SUBAPPLICATION Automatik (* Subapplication Type *)
  (* Standard: 61499-2 *)
  (* Version 1.0, 2023-01-29, Franz *)
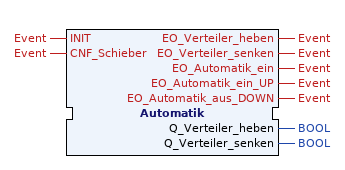
  EVENT_INPUT
    INIT;
    CNF_Schieber;
  END_EVENT
  EVENT_OUTPUT
    EO_Verteiler_heben;
    EO_Verteiler_senken;
    EO_Automatik_ein;
    EO_Automatik_ein_UP;
    EO_Automatik_aus_DOWN;
  END_EVENT
  VAR_OUTPUT
    Q_Verteiler_heben : BOOL;
    Q_Verteiler_senken : BOOL;
  END_VAR
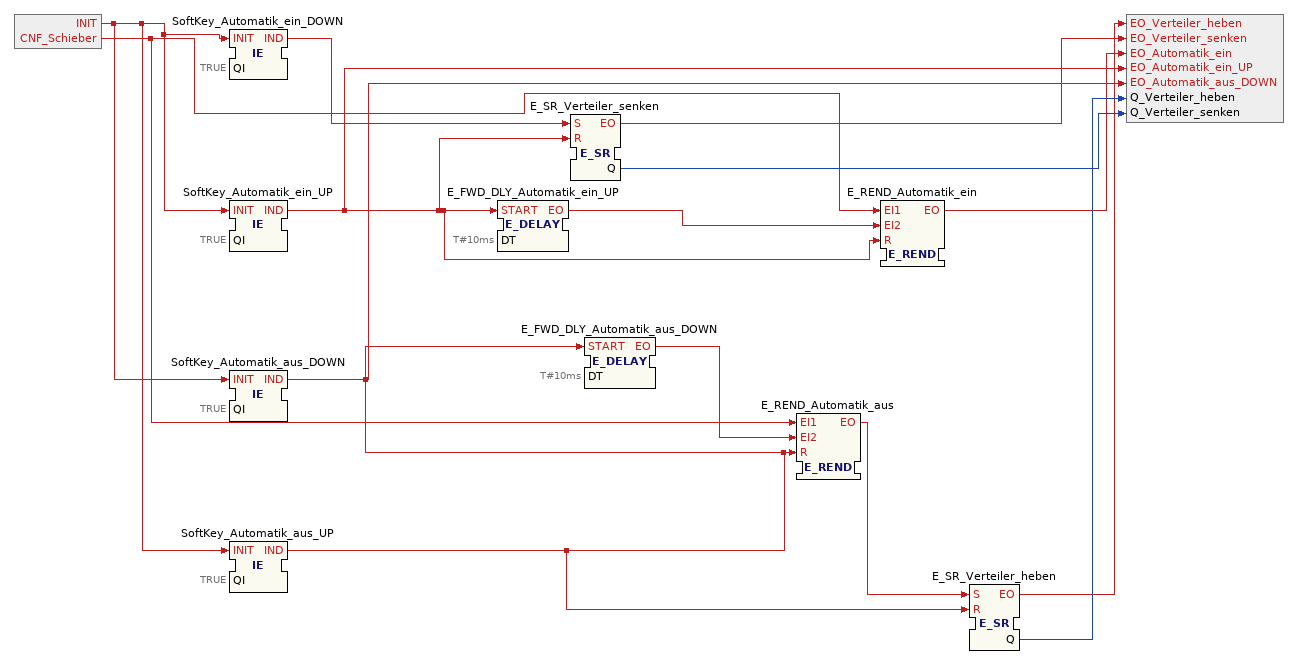
  FBS
    E_SR_Verteiler_heben : E_SR;
    E_REND_Automatik_aus : E_REND;
    E_SR_Verteiler_senken : E_SR;
    E_REND_Automatik_ein : E_REND;
    E_FWD_DLY_Automatik_ein_UP : E_DELAY(DT := T#10ms);
    E_FWD_DLY_Automatik_aus_DOWN : E_DELAY(DT := T#10ms);
    SoftKey_Automatik_ein_DOWN : IE(QI := TRUE);
    SoftKey_Automatik_ein_UP : IE(QI := TRUE);
    SoftKey_Automatik_aus_DOWN : IE(QI := TRUE);
    SoftKey_Automatik_aus_UP : IE(QI := TRUE);
  END_FBS
  EVENT_CONNECTIONS
    E_REND_Automatik_aus.EO TO E_SR_Verteiler_heben.S;
    E_SR_Verteiler_heben.EO TO EO_Verteiler_heben;
    E_SR_Verteiler_senken.EO TO EO_Verteiler_senken;
    CNF_Schieber TO E_REND_Automatik_ein.EI1;
    E_REND_Automatik_ein.EO TO EO_Automatik_ein;
    CNF_Schieber TO E_REND_Automatik_aus.EI1;
    E_FWD_DLY_Automatik_ein_UP.EO TO E_REND_Automatik_ein.EI2;
    E_FWD_DLY_Automatik_aus_DOWN.EO TO E_REND_Automatik_aus.EI2;
    INIT TO SoftKey_Automatik_ein_DOWN.INIT;
    SoftKey_Automatik_ein_DOWN.IND TO E_SR_Verteiler_senken.S;
    INIT TO SoftKey_Automatik_ein_UP.INIT;
    SoftKey_Automatik_ein_UP.IND TO E_SR_Verteiler_senken.R;
    SoftKey_Automatik_ein_UP.IND TO E_REND_Automatik_ein.R;
    SoftKey_Automatik_ein_UP.IND TO EO_Automatik_ein_UP;
    SoftKey_Automatik_ein_UP.IND TO E_FWD_DLY_Automatik_ein_UP.START;
    INIT TO SoftKey_Automatik_aus_DOWN.INIT;
    SoftKey_Automatik_aus_DOWN.IND TO E_REND_Automatik_aus.R;
    SoftKey_Automatik_aus_DOWN.IND TO EO_Automatik_aus_DOWN;
    SoftKey_Automatik_aus_DOWN.IND TO E_FWD_DLY_Automatik_aus_DOWN.START;
    INIT TO SoftKey_Automatik_aus_UP.INIT;
    SoftKey_Automatik_aus_UP.IND TO E_SR_Verteiler_heben.R;
    SoftKey_Automatik_aus_UP.IND TO E_REND_Automatik_aus.R;
  END_CONNECTIONS
  DATA_CONNECTIONS
    E_SR_Verteiler_heben.Q TO Q_Verteiler_heben;
    E_SR_Verteiler_senken.Q TO Q_Verteiler_senken;
  END_CONNECTIONS
END_SUBAPPLICATION
